Staubli VAL3: shiftArray.pgx

public program shiftArray(num& x_nNum[])
  local num l_nIndex
begin

  //shift up a 1d num array

  for l_nIndex=0 to size(x_nNum)-2
    x_nNum[l_nIndex] = x_nNum[l_nIndex+1]
  endFor

  x_nNum[size(x_nNum)-1]=0

end
